{attribute 'GeneratedUsingTerminal: EL2502-0010-0020'}
{attribute addProperty BoxType "EL2502-0010-0020"}
{attribute addProperty Id "StatusAT %I*Status_8A0522A04"}
{attribute addProperty CRC "1111094866"}
{attribute addProperty Size "4"}
TYPE PWM_Inputs_Channel_4239F652 :
STRUCT
	{attribute addProperty Name "Status"}
	Status AT %I* : Status_8A0522A0;
END_STRUCT
END_TYPE

(* stored: Version 1.2.0.0, ProductVersion 3.1.4024.9
   DUT PWM_Inputs_Channel_4239F652: Id {5ec26d79-1d39-423e-a37b-ad155a0a19b2} *)
